PROGRAM CNC_1
VAR
		

END_VAR

Servo();

END_PROGRAM

(* stored: Version 1.1.0.1, ProductVersion 3.1.4024.11
   POU CNC_1: Id {067559b7-2cc8-4a74-b07e-41eb917a7856}, SpecialFunc None *)
